// Test-only child of FB_TwoPosActuator. The production FB keeps io,
// advancePermissives, and retractPermissives in its private VAR section,
// so tests use this probe to inject field signals and map permissives
// without touching the public surface.
//
// The probe delegates the cyclic body back to the parent via SUPER^() —
// without that call the child's empty body would replace the parent's
// state-machine logic and every assertion would see zeroed state.
//
// Lives in the Testing project only — not part of TcForge's public API.
FUNCTION_BLOCK FB_TwoPosActuator_Probe EXTENDS TcForge.FB_TwoPosActuator

// Run the inherited state machine using the probe's injected signals.
SUPER^();

METHOD PUBLIC SetAdvancedFeedback
VAR_INPUT
    bValue : BOOL;
END_VAR
io.inFbkAdvanced := bValue;
END_METHOD

METHOD PUBLIC SetRetractedFeedback
VAR_INPUT
    bValue : BOOL;
END_VAR
io.inFbkRetracted := bValue;
END_METHOD

METHOD PUBLIC GetValveAdvance : BOOL
GetValveAdvance := io.outValveAdvance;
END_METHOD

METHOD PUBLIC GetValveRetract : BOOL
GetValveRetract := io.outValveRetract;
END_METHOD

// Map a single permissive bit into advancePermissives so tests can force
// REJECTED_PERMISSIVE_NOT_MET / PermissivesNotOK without touching the
// production code's permissive wiring.
METHOD PUBLIC MapAdvancePerm
VAR_INPUT
    nBit   : UDINT;
    bValue : BOOL;
END_VAR
advancePermissives.MapInput(bitIndex := nBit, inputValue := bValue);
END_METHOD

METHOD PUBLIC MapRetractPerm
VAR_INPUT
    nBit   : UDINT;
    bValue : BOOL;
END_VAR
retractPermissives.MapInput(bitIndex := nBit, inputValue := bValue);
END_METHOD

END_FUNCTION_BLOCK

(* stored: Version 1.1.0.1, ProductVersion 3.1.4026.12
   POU FB_TwoPosActuator_Probe: Id {b1c2d3e4-f5a6-7890-abcd-000000000b00}, SpecialFunc None
   Method SetAdvancedFeedback: Id {b1c2d3e4-f5a6-7890-abcd-000000000b01}
   Method SetRetractedFeedback: Id {b1c2d3e4-f5a6-7890-abcd-000000000b02}
   Method GetValveAdvance: Id {b1c2d3e4-f5a6-7890-abcd-000000000b03}
   Method GetValveRetract: Id {b1c2d3e4-f5a6-7890-abcd-000000000b04}
   Method MapAdvancePerm: Id {b1c2d3e4-f5a6-7890-abcd-000000000b05}
   Method MapRetractPerm: Id {b1c2d3e4-f5a6-7890-abcd-000000000b06} *)
